(* CoDeSys 2.3.9.41 project: Berdyansl_KNS_bez_zadv.pro *)
(* Libraries: ComService.lib 21.5.09 13:28:28, SysLibCom.lib 20.2.06 12:31:08, ModBus.lib 27.5.09 08:22:38, STANDARD.LIB 4.10.05 10:14:46, IECSFC.LIB 13.4.06 14:51:28, SYSLIBTIME.LIB 20.2.06 12:31:16, SYSTASKINFO.LIB 20.2.06 12:31:38, ANALYZATION.LIB 5.10.99 08:05:06 *)

(* PLC configuration (modules and I/O channels)
DInputs [ID10051] node 0, in %IB0.0 out %QB0.0 {BName = #NДискретные Вх.#A0}
  AT %IB0.0.0 [DInput] Битовая маска входов {CPString128 = #NСост.Дискр.Вх.#Fr.Cn#H2D26#A3#T02#O#B0120#V2; DinLM = #NЛогика Дискр.Вх#Finv.D#B0121#A0#V2#T02#D00#MFF; DinFl = #NПост.Ф.ДребКонт#FTin.F#B0122#A0#U0017#T02#D0A#MFF}
Outputs [ID10057] node 1, in %IB0.1 out %QB0.1 {BName = #NВУ#A0}
  AT %QD0.1.0 [AnalogOutput0] Выход 1 {CPString128 = #NСост.ВУ1#Fr.oe#I00#B0000#A0#O#C3#T00#M+1.00E+00; AoutPWMP = #NПериод ШИМ ВУ1#Fthpd#I00#B0123#A0#U0017#T01#D03E8#L0002#MFDE8; AoutPWMM = #NМин.имп.ШИМ ВУ1#Ft.L#I00#B012B#A0#U0017#T01#D0032#L0001#M1388; AoutSafeValue = #NБезоп.сост.ВУ1#FO.ALr#I00#B0010#A0#C3#T00#D+0.00E+00#M+1.00E+00}
  DO2 AT %QD0.1.1 [AnalogOutput1] Пуск Плавного пуска 2 {CPString128 = #NСост.ВУ2#Fr.oe#HE894#I01#A0#T00#C3#M+1.00E+00#O#B0002; AoutPWMP = #NПериод ШИМ ВУ2#Fthpd#I01#B0124#A0#U0017#T01#D03E8#L0002#MFDE8; AoutPWMM = #NМин.имп.ШИМ ВУ2#Ft.L#I01#B012C#A0#U0017#T01#D0032#L0001#M1388; AoutSafeValue = #NБезоп.сост.ВУ2#FO.ALr#I01#B0012#A0#C3#T00#D+0.00E+00#M+1.00E+00}
  DO3 AT %QD0.1.2 [AnalogOutput2] Пуск Плавного пуска 1 {CPString128 = #NСост.ВУ3#Fr.oe#HE894#I02#A0#T00#C3#M+1.00E+00#O#B0004; AoutPWMP = #NПериод ШИМ ВУ3#Fthpd#I02#B0125#A0#U0017#T01#D03E8#L0002#MFDE8; AoutPWMM = #NМин.имп.ШИМ ВУ3#Ft.L#I02#B012D#A0#U0017#T01#D0032#L0001#M1388; AoutSafeValue = #NБезоп.сост.ВУ3#FO.ALr#I02#B0014#A0#C3#T00#D+0.00E+00#M+1.00E+00}
  DO4 AT %QD0.1.3 [AnalogOutput3] Авария {CPString128 = #NСост.ВУ4#Fr.oe#HE894#I03#A0#T00#C3#M+1.00E+00#O#B0006; AoutPWMP = #NПериод ШИМ ВУ4#Fthpd#I03#B0126#A0#U0017#T01#D03E8#L0002#MFDE8; AoutPWMM = #NМин.имп.ШИМ ВУ4#Ft.L#I03#B012E#A0#U0017#T01#D0032#L0001#M1388; AoutSafeValue = #NБезоп.сост.ВУ4#FO.ALr#I03#B0016#A0#C3#T00#D+0.00E+00#M+1.00E+00}
  DO5 AT %QD0.1.4 [AnalogOutput4] Питание Видеокамеры {CPString128 = #NСост.ВУ5#Fr.oe#HE894#I04#A0#T00#C3#M+1.00E+00#O#B0008; AoutPWMP = #NПериод ШИМ ВУ5#Fthpd#I04#B0127#A0#U0017#T01#D03E8#L0002#MFDE8; AoutPWMM = #NМин.имп.ШИМ ВУ5#Ft.L#I04#B012F#A0#U0017#T01#D0032#L0001#M1388; AoutSafeValue = #NБезоп.сост.ВУ5#FO.ALr#I04#B0018#A0#C3#T00#D+0.00E+00#M+1.00E+00}
  DO6 AT %QD0.1.5 [AnalogOutput5] Управление Дренажным насосом {CPString128 = #NСост.ВУ6#Fr.oe#HE894#I05#A0#T00#C3#M+1.00E+00#O#B000A; AoutPWMP = #NПериод ШИМ ВУ6#Fthpd#I05#B0128#A0#U0017#T01#D03E8#L0002#MFDE8; AoutPWMM = #NМин.имп.ШИМ ВУ6#Ft.L#I05#A0#B0130#U0017#T01#D0032#L0001#M1388; AoutSafeValue = #NБезоп.сост.ВУ6#FO.ALr#I05#B001A#A0#C3#T00#D+0.00E+00#M+1.00E+00}
  DO7 AT %QD0.1.6 [AnalogOutput6] Управление ПЛАВНЫМ ПУСКОМ НАСОСА 2 {CPString128 = #NСост.ВУ7#Fr.oe#HE894#I06#A0#T00#C3#M+1.00E+00#O#B000C; AoutPWMP = #NПериод ШИМ ВУ7#Fthpd#I06#B0129#A0#U0017#T01#D03E8#L0002#MFDE8; AoutPWMM = #NМин.имп.ШИМ ВУ7#Ft.L#I06#B0131#A0#U0017#T01#D0032#L0001#M1388; AoutSafeValue = #NБезоп.сост.ВУ7#FO.ALr#I06#B001C#A0#C3#T00#D+0.00E+00#M+1.00E+00}
  DO8 AT %QD0.1.7 [AnalogOutput7] Управление ПЛАВНЫМ ПУСКОМ НАСОСА 1 {CPString128 = #NСост.ВУ8#Fr.oe#HE894#I07#A0#T00#C3#M+1.00E+00#O#B000E; AoutPWMP = #NПериод ШИМ ВУ8#Fthpd#I07#B012A#A0#U0017#T01#D03E8#L0002#MFDE8; AoutPWMM = #NМин.имп.ШИМ ВУ8#Ft.L#I07#A0#B0132#U0017#T01#D0032#L0001#M1388; AoutSafeValue = #NБезоп.сост.ВУ8#FO.ALr#I07#B001E#A0#C3#T00#D+0.00E+00#M+1.00E+00}
AInputs [ID10055] node 2, in %IB0.2 out %QB0.2 {BName = #NАналоговые Вх.#A0; Spay = #NКоррекция ХС#Fcj-.c#B0133#A0#U002A#T03#D01}
  AT %ID0.2.0 [AnalogInput0] Аналоговый вход 1 {CPString128 = #NДатчик уровня#Fread#H8784#I00#A3#T10#C2#O#B0020#V3; AinType = #NТип датчика 1#Fin-t#H932D#I00#A0#U002F#T04#D10#M15#B0134; InFD = #NПост. фильтра 1#Fin.Fd#I00#B013C#A0#U0018#T01#D0005#M0708; InFG = #NПолоса Фильтра1#Fin.FG#I00#B0030#A0#T00#D+1.00E+01#L+0.00E+01#M+9.99E+03}
  AT %ID0.2.1 [AnalogInputTime0] Время измерения 1
  AI AT %ID0.2.2 [AnalogInput1] Аналоговый вход 2 {CPString128 = #NДатчик давления#Fread#H8784#I01#A3#T10#C2#O#B0022#V3; AinType = #NДатчик уровня#Fin-t#H932D#I01#A0#U002F#T04#D10#M15#B0135; InFD = #NПост. фильтра 2#Fin.Fd#H1659#I01#A0#U0018#T01#D0005#M0708#B013D; InFG = #NПолоса Фильтра2#Fin.FG#I01#B0032#A0#T00#D+1.00E+01#L+0.00E+01#M+9.99E+03}
  AT %ID0.2.3 [AnalogInputTime1] Время измерения 2
  AT %ID0.2.4 [AnalogInput2] Аналоговый вход 3 {CPString128 = #NВход 3#Fread#H8784#I02#A3#T10#C2#O#B0024#V3; AinType = #NТип датчика 3#Fin-t#H932D#I02#A0#U002F#T04#D00#M15#B0136; InFD = #NПост. фильтра 3#Fin.Fd#I02#B013E#A0#U0018#T01#D0005#M0708; InFG = #NПолоса Фильтра3#Fin.FG#I02#B0034#A0#T00#D+1.00E+01#L+0.00E+01#M+9.99E+03}
  AT %ID0.2.5 [AnalogInputTime2] Время измерения 3
  AT %ID0.2.6 [AnalogInput3] Аналоговый вход 4 {CPString128 = #NВход 4#Fread#H8784#I03#A3#T10#C2#O#B0026#V3; AinType = #NТип датчика 4#Fin-t#H932D#I03#A0#U002F#T04#D00#M15#B0137; InFD = #NПост. фильтра 4#Fin.Fd#I03#B013F#A0#U0018#T01#D0005#M0708; InFG = #NПолоса Фильтра4#Fin.FG#I03#A0#B0036#T00#D+1.00E+01#L+0.00E+01#M+9.99E+03}
  AT %ID0.2.7 [AnalogInputTime3] Время измерения 4
  AT %ID0.2.8 [AnalogInput4] Аналоговый вход 5 {CPString128 = #NВход 5#Fread#H8784#I04#A3#T10#C2#O#B0028#V3; AinType = #NТип датчика 5#Fin-t#H932D#I04#A0#U002F#T04#D00#M15#B0138; InFD = #NПост. фильтра 5#Fin.Fd#I04#B0140#A0#U0018#T01#D0005#M0708; InFG = #NПолоса Фильтра5#Fin.FG#I04#B0038#A0#T00#D+1.00E+01#L+0.00E+01#M+9.99E+03}
  AT %ID0.2.9 [AnalogInputTime4] Время измерения 5
  AT %ID0.2.10 [AnalogInput5] Аналоговый вход 6 {CPString128 = #NВход 6#Fread#H8784#I05#A3#T10#C2#O#B002A#V3; AinType = #NТип датчика 6#Fin-t#H932D#I05#A0#U002F#T04#D00#M15#B0139; InFD = #NПост. фильтра 6#Fin.Fd#I05#B0141#A0#U0018#T01#D0005#M0708; InFG = #NПолоса Фильтра6#Fin.FG#I05#B003A#A0#T00#D+1.00E+01#L+0.00E+01#M+9.99E+03}
  AT %ID0.2.11 [AnalogInputTime5] Время измерения 6
  AT %ID0.2.12 [AnalogInput6] Аналоговый вход 7 {CPString128 = #NВход 7#Fread#H8784#I06#A3#T10#C2#O#B002C#V3; AinType = #NТип датчика 7#Fin-t#H932D#I06#A0#U002F#T04#D00#M15#B013A; InFD = #NПост. фильтра 7#Fin.Fd#I06#B0142#A0#U0018#T01#D0005#M0708; InFG = #NПолоса Фильтра7#Fin.FG#I06#B003C#A0#T00#D+1.00E+01#L+0.00E+01#M+9.99E+03}
  AT %ID0.2.13 [AnalogInputTime6] Время измерения 7
  AT %ID0.2.14 [AnalogInput7] Аналоговый вход 8 {CPString128 = #NВход 8#Fread#H8784#I07#A3#T10#C2#O#B002E#V3; AinType = #NТип датчика 8#Fin-t#H932D#I07#A0#U002F#T04#D00#M15#B013B; InFD = #NПост. фильтра 8#Fin.Fd#I07#B0143#A0#U0018#T01#D0005#M0708; InFG = #NПолоса Фильтра8#Fin.FG#I07#B003E#A0#T00#D+1.00E+01#L+0.00E+01#M+9.99E+03}
  AT %ID0.2.15 [AnalogInputTime7] Время измерения 8
MR1_Outputs [ID10053] node 3, in %IB0.3 out %QB0.3 {BName = #NВУ МР1#A0}
  AT %QB0.3.0 [DOutput] ВУ МР1 {CPString128 = #NСост.ВУ МР1#Fr.oe.s#B0144#A0#O#V2#T02}
Additional [ID10059] node 4, in %IB0.4 out %QB0.4 {BName = #NДоп.пар-ры#A0}
  Illumination AT %QB0.4.0 [LCDLight] Подсветка {CPString128 = #NЯрк.подсв.ЖКИ#Find.i#H1845#A0#T02#D2D#M32#B0145}
  AT %QB0.4.1 [LCDContrast] Контраст {CPString128 = #NКонтраст ЖКИ#Find.C#H074A#A0#T02#D19#M20#L05#B0146}
  Keyboard AT %IW0.4.2 [KBD] Клавиатура {CPString128 = #NСост.клавиатуры#Fkbrd#H399B#A3#T02#O#B0147; KBDBeep = #NЗвук кнопок#Fbeep#B0148#A0#U002A#T03#D01}
  Clock AT %QD0.4.3 [RTS] Часы контроллера {RTSPar = #NВремя и дата#FrtC#HFA30#A0#T05#O#B0040}
  Svetodiod AT %QB0.4.4 [LED] Светодиоды {CPString128 = #NСос.светодиодов#Find.L#HF304#A0#T02#D00#M3F#L00#O#B0149#V2}
Versions [ID10060] node 5, in %IB0.5 out %QB0.5 {BName = #NВерсииПрошивок#A0}
  AT %QB0.5.0 [DevName] Имя устройства {CPString128 = #NИмя устройства#Fdev#B0042#A3#O#T08}
  AT %IB0.5.1 [HardVer] Прошивка {CPString128 = #NВерсия прошивки#Fver#B004A#A3#O#T08}
  AT %QB0.5.2 [SoftVer] Программа {CPString128 = #NВерсияПрограммы#Fp.ver#B0052#A3#O#T08}
RS-1 [ID10061] node 6, in %IB0.6 out %QB0.6 {BName = #NНастр.RS-1#A0; RSBPS = #NСкорость#FbPS#I00#B014A#A0#U0046#T04#D00#M09; RSWLen = #NДлина слова#FLen#I00#B014B#A0#U0005#T04#D03#M03; RSPrt = #NЧётность#Fprty#I00#B014C#A0#U009A#T04#D04#M04; RSStp = #NСтоп биты#Fsbit#I00#B014D#A0#U00A1#T04#D00#M02; RSALen = #NДлина адреса#Fa.len#I00#B014E#A0#U0055#T03#D00; RSAdr = #NАдрес прибора#FAddr#I00#B014F#A0#T01#D0010#M07FF; RSDl = #NЗадержка ответа#FRs.dl#I00#B0150#A0#U0017#T02#D05#M32}
RS-2 [ID10062] node 7, in %IB0.7 out %QB0.7 {BName = #NНастр.RS-2#A0; RSBPS = #NСкорость#FbPS#I01#B0151#A0#U0046#T04#D00#M09; RSWLen = #NДлина слова#FLen#I01#B0152#A0#U0005#T04#D03#M03; RSPrt = #NЧётность#Fprty#I01#B0153#A0#U009A#T04#D04#M04; RSStp = #NСтоп биты#Fsbit#I01#B0154#A0#U00A1#T04#D00#M02; RSALen = #NДлина адреса#Fa.len#I01#B0155#A0#U0055#T03#D00; RSAdr = #NАдрес прибора#FAddr#I01#B0156#A0#T01#D0010#M07FF; RSDl = #NЗадержка ответа#FRs.dl#I01#B0157#A0#U0017#T02#D05#M32}
WorkInd [ID10100] node 1, in %IB1 out %QB1 {WIChanelCount = 6}
SubMenu [ID11000] node 2, in %IB2 out %QB2 {BName = #NВетка#A0}
  SubMenu [ID11000] node 0, in %IB2.0 out %QB2.0 {BName = #NВетка#A0}
ATS22_1_p84 AT %QX2.0.0.0 [BoolPar] Канал управления Mb\клемник {CPString128 = #NБулевский#A0#U00AA#T03#D00}
ATS22_1_p752b3 AT %QX2.0.1.0 [BoolPar] Сброс Аварии {CPString128 = #NБулевский#A0#U00AA#T03#D00}
SubMenu [ID11000] node 1, in %IB2.1 out %QB2.1 {BName = #NВетка#A0}
mb_in1 AT %QX2.1.0.0 [BoolPar] {CPString128 = #NБулевский#A0#U00AA#T03#D00#O}
mb_in2 AT %QX2.1.1.0 [BoolPar] {CPString128 = #NБулевский#A0#U00AA#T03#D00#O}
mb_in3 AT %QX2.1.2.0 [BoolPar] {CPString128 = #NБулевский#A0#U00AA#T03#D00#O}
mb_in4 AT %QX2.1.3.0 [BoolPar] {CPString128 = #NБулевский#A0#U00AA#T03#D00#O}
mb_in5 AT %QX2.1.4.0 [BoolPar] {CPString128 = #NБулевский#A0#U00AA#T03#D00}
mb_in6 AT %QX2.1.5.0 [BoolPar] {CPString128 = #NБулевский#A0#U00AA#T03#D00}
mb_in7 AT %QX2.1.6.0 [BoolPar] {CPString128 = #NБулевский#A0#U00AA#T03#D00}
mb_in8 AT %QX2.1.7.0 [BoolPar] {CPString128 = #NБулевский#A0#U00AA#T03#D00}
mb_in9 AT %QX2.1.8.0 [BoolPar] {CPString128 = #NБулевский#A0#U00AA#T03#D00}
mb_in10 AT %QX2.1.9.0 [BoolPar] {CPString128 = #NБулевский#A0#U00AA#T03#D00}
mb_in11 AT %QX2.1.10.0 [BoolPar] {CPString128 = #NБулевский#A0#U00AA#T03#D00}
mb_in12 AT %QX2.1.11.0 [BoolPar] {CPString128 = #NБулевский#A0#U00AA#T03#D00}
mb_in13 AT %QX2.1.12.0 [BoolPar] Контроль доступа Датч 1 {CPString128 = #NБулевский#A0#U00AA#T03#D00}
mb_in14 AT %QX2.1.13.0 [BoolPar] {CPString128 = #NБулевский#A0#U00AA#T03#D00}
mb_in15 AT %QX2.1.14.0 [BoolPar] {CPString128 = #NБулевский#A0#U00AA#T03#D00}
mb_in16 AT %QX2.1.15.0 [BoolPar] {CPString128 = #NБулевский#A0#U00AA#T03#D00}
mb_in17 AT %QX2.1.16.0 [BoolPar] {CPString128 = #NБулевский#A0#U00AA#T03#D00}
mb_in18 AT %QX2.1.17.0 [BoolPar] {CPString128 = #NБулевский#A0#U00AA#T03#D00}
mb_in19 AT %QX2.1.18.0 [BoolPar] {CPString128 = #NБулевский#A0#U00AA#T03#D00}
mb_in20 AT %QX2.1.19.0 [BoolPar] {CPString128 = #NБулевский#A0#U00AA#T03#D00}
mb_in21 AT %QX2.1.20.0 [BoolPar] {CPString128 = #NБулевский#A0#U00AA#T03#D00}
mb_in22 AT %QX2.1.21.0 [BoolPar] {CPString128 = #NБулевский#A0#U00AA#T03#D00}
mb_in23 AT %QX2.1.22.0 [BoolPar] {CPString128 = #NБулевский#A0#U00AA#T03#D00}
mb_in24 AT %QX2.1.23.0 [BoolPar] {CPString128 = #NБулевский#A0#U00AA#T03#D00}
%Mmb_in25 AT %QX2.1.24.0 [BoolPar] {CPString128 = #NБулевский#A0#U00AA#T03#D00}
mb_in26 AT %QX2.1.25.0 [BoolPar] {CPString128 = #NБулевский#A0#U00AA#T03#D00}
mb_in27 AT %QX2.1.26.0 [BoolPar] {CPString128 = #NБулевский#A0#U00AA#T03#D00}
mb_in28 AT %QX2.1.27.0 [BoolPar] {CPString128 = #NБулевский#A0#U00AA#T03#D00}
mb_in29 AT %QX2.1.28.0 [BoolPar] {CPString128 = #NБулевский#A0#U00AA#T03#D00}
mb_in30 AT %QX2.1.29.0 [BoolPar] {CPString128 = #NБулевский#A0#U00AA#T03#D00}
mb_in31 AT %QX2.1.30.0 [BoolPar] {CPString128 = #NБулевский#A0#U00AA#T03#D00}
mb_in32 AT %QX2.1.31.0 [BoolPar] {CPString128 = #NБулевский#A0#U00AA#T03#D00}
ATS22_2_p84 AT %QX2.2.0.0 [BoolPar] Канал управления Mb\клемник {CPString128 = #NБулевский#A0#U00AA#T03#D00}
ATS22_2_p752b3 AT %QX2.2.1.0 [BoolPar] Сброс Аварии {CPString128 = #NБулевский#A0#U00AA#T03#D00}
ubz_1_p100 AT %QW3.0.0.0 [IntPar] Ток А {CPString128 = #NЦелое#A0#T01#D0000}
ubz_1_p101 AT %QW3.0.1.0 [IntPar] Ток В {CPString128 = #NЦелое#A0#T01#D0000}
ubz_1_p102 AT %QW3.0.2.0 [IntPar] Ток С {CPString128 = #NЦелое#A0#T01#D0000}
ubz_1_p103 AT %QW3.0.3.0 [IntPar] Ток нулевой последовательности {CPString128 = #NЦелое#A0#T01#D0000}
ubz_1_p113 AT %QW3.0.4.0 [IntPar] {CPString128 = #NЦелое#A0#T01#D0000}
ubz_1_p114 AT %QW3.0.5.0 [IntPar] {CPString128 = #NЦелое#A0#T01#D0000}
ubz_1_p115 AT %QW3.0.6.0 [IntPar] {CPString128 = #NЦелое#A0#T01#D0000}
ubz_1_p116 AT %QW3.0.7.0 [IntPar] {CPString128 = #NЦелое#A0#T01#D0000}
ubz_1_p117 AT %QW3.0.8.0 [IntPar] Линейное напряжение А {CPString128 = #NЦелое#A0#T01#D0000}
ubz_1_p118 AT %QW3.0.9.0 [IntPar] {CPString128 = #NЦелое#A0#T01#D0000}
ubz_1_p119 AT %QW3.0.10.0 [IntPar] {CPString128 = #NЦелое#A0#T01#D0000}
ubz_1_p120 AT %QW3.0.11.0 [IntPar] {CPString128 = #NЦелое#A0#T01#D0000}
ubz_1_p121 AT %QW3.0.12.0 [IntPar] {CPString128 = #NЦелое#A0#T01#D0000}
ubz_1_p122 AT %QW3.0.13.0 [IntPar] {CPString128 = #NЦелое#A0#T01#D0000}
IntP [ID11200] node 14, in %IB3.0.14 out %QB3.0.14
  ubz_1_p241 AT %QW3.0.14.0 [IntPar] {CPString128 = #NЦелое#A0#T01#D0000}
IntP [ID11200] node 15, in %IB3.0.15 out %QB3.0.15
  ubz_1_p242 AT %QW3.0.15.0 [IntPar] {CPString128 = #NЦелое#A0#T01#D0000}
ubz_1_p240 AT %QB3.0.16.0 [BytePar] Регистр состояния УБЗ {CPString128 = #NБайт#A0#T02#D00}
ubz_1_p241_1 AT %QB3.0.17.0 [BytePar] Регистр Аварии 1 {CPString128 = #NБайт#A0#T02#D00}
ubz_1_p241_2 AT %QB3.0.18.0 [BytePar] Регистр Аварии 1 {CPString128 = #NБайт#A0#T02#D00}
ubz_1_p242_1 AT %QB3.0.19.0 [BytePar] Регистр Аварии 2 {CPString128 = #NБайт#A0#T02#D00}
ubz_1_p242_2 AT %QB3.0.20.0 [BytePar] Регистр Аварии 2 {CPString128 = #NБайт#A0#T02#D00}
SubMenu [ID11000] node 1, in %IB3.1 out %QB3.1 {BName = #NВетка#A0}
ubz_2_p100 AT %QW3.1.0.0 [IntPar] Ток А {CPString128 = #NЦелое#A0#T01#D0000}
ubz_2_p101 AT %QW3.1.1.0 [IntPar] Ток В {CPString128 = #NЦелое#A0#T01#D0000}
ubz_2_p102 AT %QW3.1.2.0 [IntPar] Ток С {CPString128 = #NЦелое#A0#T01#D0000}
ubz_2_p103 AT %QW3.1.3.0 [IntPar] Ток нулевой последовательности {CPString128 = #NЦелое#A0#T01#D0000}
ubz_2_p113 AT %QW3.1.4.0 [IntPar] {CPString128 = #NЦелое#A0#T01#D0000}
ubz_2_p114 AT %QW3.1.5.0 [IntPar] {CPString128 = #NЦелое#A0#T01#D0000}
ubz_2_p115 AT %QW3.1.6.0 [IntPar] {CPString128 = #NЦелое#A0#T01#D0000}
ubz_2_p116 AT %QW3.1.7.0 [IntPar] {CPString128 = #NЦелое#A0#T01#D0000}
ubz_2_p117 AT %QW3.1.8.0 [IntPar] Линейное напряжение А {CPString128 = #NЦелое#A0#T01#D0000}
ubz_2_p118 AT %QW3.1.9.0 [IntPar] {CPString128 = #NЦелое#A0#T01#D0000}
ubz_2_p119 AT %QW3.1.10.0 [IntPar] {CPString128 = #NЦелое#A0#T01#D0000}
ubz_2_p120 AT %QW3.1.11.0 [IntPar] {CPString128 = #NЦелое#A0#T01#D0000}
ubz_2_p121 AT %QW3.1.12.0 [IntPar] {CPString128 = #NЦелое#A0#T01#D0000}
ubz_2_p122 AT %QW3.1.13.0 [IntPar] {CPString128 = #NЦелое#A0#T01#D0000}
IntP [ID11200] node 14, in %IB3.1.14 out %QB3.1.14
  ubz_2_p241 AT %QW3.1.14.0 [IntPar] {CPString128 = #NЦелое#A0#T01#D0000}
  ubz_2_p242 AT %QW3.1.15.0 [IntPar] {CPString128 = #NЦелое#A0#T01#D0000}
SubMenu [ID11000] node 2, in %IB3.2 out %QB3.2 {BName = #NВетка#A0}
ATS22_1_p279 AT %QW3.2.0.0 [IntPar] Проследняя неисправность {CPString128 = #NЦелое#A0#T01#D0000}
ATS22_1_p256 AT %QW3.2.1.0 [IntPar] Состояние Плавноо пуска {CPString128 = #NЦелое#A0#T01#D0000}
ATS22_1_p257 AT %QW3.2.2.0 [IntPar] Ток фазы А {CPString128 = #NЦелое#A0#T01#D0000}
ATS22_1_p259 AT %QW3.2.3.0 [IntPar] Ток фазы С {CPString128 = #NЦелое#A0#T01#D0000}
ATS22_1_p258 AT %QW3.2.4.0 [IntPar] Ток фазы В {CPString128 = #NЦелое#A0#T01#D0000}
ATS22_1_p260 AT %QW3.2.5.0 [IntPar] Линейное напряжение {CPString128 = #NЦелое#A0#T01#D0000}
SubMenu [ID11000] node 3, in %IB3.3 out %QB3.3 {BName = #NВетка#A0}
ATS22_2_p279 AT %QW3.3.0.0 [IntPar] {CPString128 = #NЦелое#A0#T01#D0000}
ATS22_2_p256 AT %QW3.3.1.0 [IntPar] {CPString128 = #NЦелое#A0#T01#D0000}
ATS22_2_p257 AT %QW3.3.2.0 [IntPar] {CPString128 = #NЦелое#A0#T01#D0000}
ATS22_2_p259 AT %QW3.3.3.0 [IntPar] {CPString128 = #NЦелое#A0#T01#D0000}
ATS22_2_p258 AT %QW3.3.4.0 [IntPar] {CPString128 = #NЦелое#A0#T01#D0000}
ATS22_2_p260 AT %QW3.3.5.0 [IntPar] {CPString128 = #NЦелое#A0#T01#D0000}
SubMenu [ID11000] node 4, in %IB4 out %QB4 {BName = #NВетка#A0}
*)

(* Global variable list: Global_Variables *)
VAR_GLOBAL
(*+++++++++++++++++++++++++++++++++++++++++++++++++++++++++++++++++++*)
(* переменные Modbus *)
	funcComService:COM_SERVICE;(*экземпляр COM_SERVICE*)
	cmSettings:COMSETTINGS;(* настройки COM- порта *)
	cmpl: BOOL;(* статус выполнения*)
	Buffer:ARRAY[0..255] OF BYTE;								(*буфер данных Modbus*)

(*+++++++++++++++++++++++++++++++++++++++++++++++++++++++++++++++++++*)

(*+++++++++++++++++++++++++++++++++++++++++++++++++++++++++++++++++++*)
(* Переменные плавного пуска №1*)
	Status_UZ1:WORD; (* Состояние плавного пуска №1 *)

(* Переменные плавного пуска №2*)
	Status_UZ2:WORD; (* Состояние плавного пуска №2 *)

(* Переменные УБЗ-302 №1 *)
	Alarm_UBZ1_p241:WORD; (*Аварии двигателя  УБЗ*)
	Alarm_UBZ1_p242:WORD; (*Аварии самого УБЗ*)

END_VAR

(* POU PLC_PRG, ST *)
PROGRAM PLC_PRG
VAR
END_VAR
prgModbus();
END_PROGRAM

(* POU prgModbus, ST *)
PROGRAM prgModbus
VAR

	byMbRequest:BYTE:=0;(* Номер опроса по Мб *)
	funcMbReadHoldRegs:MB_RD_HOLD_REGS;(*Modbus, экземпляр функ. 03, чтение регистров хранения*)
	funcMbReadInpRegs:MB_RD_INP_REGS;(*Modbus, экземпляр функ. 04, чтение регистров ввода*)
	funcMbWriteSngReg:MB_WR_SNG_REG;(*Modbus, экземпляр функ. 06, запись регистра хранения*)
	funcMbWriteRegs:MB_WR_REGS;(*Modbus, экземпляр функ. 16, запись регистров хранения*)


END_VAR
(* Обработка данных Modbus *)
	IF NOT funcComService.ready THEN
		cmSettings.Port:=1;(*номер COM-порта*)
		cmSettings.dwBaudRate:=19200;
		cmSettings.byParity:=0;
		cmSettings.dwTimeout:=0;
		cmSettings.byStopBits:=0;
		cmSettings.dwBufferSize:=0;
		cmSettings.dwScan:=0;
		funcComService(Enable:=TRUE , Settings:=cmSettings , Task:=OPEN_TSK  );
	END_IF

(*=======================================================================*)
(*===========Опрос===============*)
IF funcComService.ready THEN
	CASE byMbRequest OF
(* Опрос UZ1 *)
(*
Add: 1;
ctrl: LCL;
tt: 5.0;
For: 8n1;
tbr 19.2;
*)
    
0:(*считывает значение состояния плавного пуска*)
			funcMbReadHoldRegs(
				Enable:=TRUE ,					(*запустить блок*)
				Mode:=MB_RTU ,				(*режим передачи*)
				DevAddr:=1 ,						(*адрес опрашиваемого устройства*)
				FirstAddr:=256 ,				(*номер регистра*)
				Quantity:=1,						(*количество регистров*)
				ComHandle:=cmSettings.Port ,
				TimeOut:=T#50ms ,				(*таймаут*)
				Buffer:=Buffer);
				IF funcMbReadHoldRegs.Complete THEN
					IF funcMbReadHoldRegs.Exception=0 THEN
						Status_UZ1:=WORD_TO_INT(BYTE_TO_WORD(Buffer[1]) OR SHL(BYTE_TO_WORD(Buffer[0]),8));
						IF Status_UZ1.0=1 THEN ATS22_1_p256:=0; (* 0 - остановлен*)
						ELSIF Status_UZ1.1=1 THEN ATS22_1_p256:=1; (* 1 - запущен*)
						ELSIF Status_UZ1.2=1 THEN ATS22_1_p256:=2; (* 3 -авария*)
						ELSIF Status_UZ1.15=1 THEN ATS22_1_p256:=3; (* 2 - плавный запуск или останов *)
						END_IF
					byMbRequest:=1;
					END_IF
				END_IF
1: (*считывает проследнюю неисправность *)
			funcMbReadHoldRegs(
				Enable:=TRUE ,					(*запустить блок*)
				Mode:=MB_RTU ,					(*режим передачи*)
				DevAddr:=1 ,						(*адрес опрашиваемого устройства*)
				FirstAddr:=279,					(*номер регистра*)
				Quantity:=1,						(*количество регистров*)
				ComHandle:=cmSettings.Port ,
				TimeOut:=T#50ms ,				(*таймаут*)
				Buffer:=Buffer);
				IF funcMbReadHoldRegs.Complete THEN
					IF funcMbReadHoldRegs.Exception=0 THEN
						ATS22_1_p279:=WORD_TO_INT(BYTE_TO_WORD(BUFFER[1]) OR SHL(BYTE_TO_WORD(BUFFER[0]),8));

						byMbRequest:=2;
					END_IF
				END_IF

2: (*считывает Ток фазы А *)
				funcMbReadHoldRegs(
				Enable:=TRUE ,					(*запустить блок*)
				Mode:=MB_RTU ,					(*режим передачи*)
				DevAddr:=1 ,						(*адрес опрашиваемого устройства*)
				FirstAddr:=257,					(*номер регистра*)
				Quantity:=1,						(*количество регистров*)
				ComHandle:=cmSettings.Port ,
				TimeOut:=T#50ms ,				(*таймаут*)
				Buffer:=Buffer);
				IF funcMbReadHoldRegs.Complete THEN
					IF funcMbReadHoldRegs.Exception=0 THEN
					ATS22_1_p257:=WORD_TO_INT(BYTE_TO_WORD(Buffer[1]) OR SHL(BYTE_TO_WORD(Buffer[0]),8));

					byMbRequest:=3;
					END_IF
				END_IF

3: (*считывает Ток фазы B *)
				funcMbReadHoldRegs(
				Enable:=TRUE ,					(*запустить блок*)
				Mode:=MB_RTU ,					(*режим передачи*)
				DevAddr:=1 ,						(*адрес опрашиваемого устройства*)
				FirstAddr:=258,					(*номер регистра*)
				Quantity:=1,						(*количество регистров*)
				ComHandle:=cmSettings.Port ,
				TimeOut:=T#50ms ,				(*таймаут*)
				Buffer:=Buffer);
				IF funcMbReadHoldRegs.Complete THEN
					IF funcMbReadHoldRegs.Exception=0 THEN
					ATS22_1_p258:=WORD_TO_INT(BYTE_TO_WORD(Buffer[1]) OR SHL(BYTE_TO_WORD(Buffer[0]),8));

					byMbRequest:=4;
					END_IF
				END_IF

4:(*считывает Ток фазы C *)
				funcMbReadHoldRegs(
				Enable:=TRUE ,					(*запустить блок*)
				Mode:=MB_RTU ,					(*режим передачи*)
				DevAddr:=1 ,						(*адрес опрашиваемого устройства*)
				FirstAddr:=259,					(*номер регистра*)
				Quantity:=1,						(*количество регистров*)
				ComHandle:=cmSettings.Port ,
				TimeOut:=T#50ms ,				(*таймаут*)
				Buffer:=Buffer);
				IF funcMbReadHoldRegs.Complete THEN
					IF funcMbReadHoldRegs.Exception=0 THEN
					ATS22_1_p259:=WORD_TO_INT(BYTE_TO_WORD(Buffer[1]) OR SHL(BYTE_TO_WORD(Buffer[0]),8));

					byMbRequest:=5;
					END_IF
				END_IF

5:	(*считывает Линейное напряжение *)
				funcMbReadHoldRegs(
				Enable:=TRUE ,					(*запустить блок*)
				Mode:=MB_RTU ,					(*режим передачи*)
				DevAddr:=1 ,						(*адрес опрашиваемого устройства*)
				FirstAddr:=260,					(*номер регистра*)
				Quantity:=1,						(*количество регистров*)
				ComHandle:=cmSettings.Port ,
				TimeOut:=T#50ms ,				(*таймаут*)
				Buffer:=Buffer);
				IF funcMbReadHoldRegs.Complete THEN
					IF funcMbReadHoldRegs.Exception=0 THEN
					ATS22_1_p260:=WORD_TO_INT(BYTE_TO_WORD(Buffer[1]) OR SHL(BYTE_TO_WORD(Buffer[0]),8));

					byMbRequest:=6;
					END_IF
				END_IF

6:	IF ATS22_1_p84 THEN (*перевод в управление по МВ*)

		funcMbWriteSngReg(
				Enable:=TRUE ,					(*запустить блок*)
				Mode:=MB_RTU ,					(*режим передачи*)
				DevAddr:=1 ,						(*адрес опрашиваемого устройства*)
				REGAddr:=84,					(*номер регистра*)
				Value:=1,						 (* Если 1 то управление по modbus *)
				ComHandle:=cmSettings.Port ,
				TimeOut:=T#20ms);
				IF funcMbWriteSngReg.Complete THEN
					byMbRequest:=7;
				END_IF
	ELSE
		funcMbWriteSngReg(
				Enable:=TRUE ,					(*запустить блок*)
				Mode:=MB_RTU ,					(*режим передачи*)
				DevAddr:=1 ,						(*адрес опрашиваемого устройства*)
				REGAddr:=84,					(*номер регистра*)
				Value:=0,						 (* Если 1 то управление по modbus *)
				ComHandle:=cmSettings.Port ,
				TimeOut:=T#20ms);
				IF funcMbWriteSngReg.Complete THEN
					byMbRequest:=7;
				END_IF
	END_IF

7: (*Сброс Аварии ATS22 №1*)
	IF ATS22_1_p752b3 THEN
		funcMbWriteSngReg(
				Enable:=TRUE ,					(*запустить блок*)
				Mode:=MB_RTU ,					(*режим передачи*)
				DevAddr:=1 ,						(*адрес опрашиваемого устройства*)
				REGAddr:=752,					(*номер регистра*)
				Value:=8,						 (* Если 1 то управление по modbus *)
				ComHandle:=cmSettings.Port ,
				TimeOut:=T#20ms);
				IF funcMbWriteSngReg.Complete THEN
					byMbRequest:=8;
				END_IF
	END_IF

(*=======================================================================*)
(* Опрос UZ2 *)
(*
Add: 2;
ctrl: LCL;
tt: 5.0;
For: 8n1;
tbr 19.2;
*)

8:(*считывает значение состояния плавного пуска*)
			funcMbReadHoldRegs(
				Enable:=TRUE ,					(*запустить блок*)
				Mode:=MB_RTU ,				(*режим передачи*)
				DevAddr:=2 ,						(*адрес опрашиваемого устройства*)
				FirstAddr:=256 ,				(*номер регистра*)
				Quantity:=1,						(*количество регистров*)
				ComHandle:=cmSettings.Port ,
				TimeOut:=T#50ms ,				(*таймаут*)
				Buffer:=Buffer);
				IF funcMbReadHoldRegs.Complete THEN
					IF funcMbReadHoldRegs.Exception=0 THEN
						Status_UZ2:=WORD_TO_INT(BYTE_TO_WORD(Buffer[1]) OR SHL(BYTE_TO_WORD(Buffer[0]),8));
						IF Status_UZ2.0=1 THEN ATS22_2_p256:=0; (* 0 - остановлен*)
						ELSIF Status_UZ2.1=1 THEN ATS22_2_p256:=1; (* 1 - запущен*)
						ELSIF Status_UZ2.2=1 THEN ATS22_2_p256:=2; (* 3 -авария*)
						ELSIF Status_UZ2.15=1 THEN ATS22_2_p256:=3; (* 2 - плавный запуск или останов *)
						END_IF
					byMbRequest:=9;
					END_IF
				END_IF
9: (*считывает проследнюю неисправность *)
			funcMbReadHoldRegs(
				Enable:=TRUE ,					(*запустить блок*)
				Mode:=MB_RTU ,					(*режим передачи*)
				DevAddr:=2 ,						(*адрес опрашиваемого устройства*)
				FirstAddr:=279,					(*номер регистра*)
				Quantity:=1,						(*количество регистров*)
				ComHandle:=cmSettings.Port ,
				TimeOut:=T#50ms ,				(*таймаут*)
				Buffer:=Buffer);
				IF funcMbReadHoldRegs.Complete THEN
					IF funcMbReadHoldRegs.Exception=0 THEN
						ATS22_2_p279:=WORD_TO_INT(BYTE_TO_WORD(BUFFER[1]) OR SHL(BYTE_TO_WORD(BUFFER[0]),8));

						byMbRequest:=10;
					END_IF
				END_IF

10: (*считывает Ток фазы А *)
				funcMbReadHoldRegs(
				Enable:=TRUE ,					(*запустить блок*)
				Mode:=MB_RTU ,					(*режим передачи*)
				DevAddr:=2 ,						(*адрес опрашиваемого устройства*)
				FirstAddr:=257,					(*номер регистра*)
				Quantity:=1,						(*количество регистров*)
				ComHandle:=cmSettings.Port ,
				TimeOut:=T#50ms ,				(*таймаут*)
				Buffer:=Buffer);
				IF funcMbReadHoldRegs.Complete THEN
					IF funcMbReadHoldRegs.Exception=0 THEN
					ATS22_2_p257:=WORD_TO_INT(BYTE_TO_WORD(Buffer[1]) OR SHL(BYTE_TO_WORD(Buffer[0]),8));

					byMbRequest:=11;
					END_IF
				END_IF

11: (*считывает Ток фазы B *)
				funcMbReadHoldRegs(
				Enable:=TRUE ,					(*запустить блок*)
				Mode:=MB_RTU ,					(*режим передачи*)
				DevAddr:=2 ,						(*адрес опрашиваемого устройства*)
				FirstAddr:=258,					(*номер регистра*)
				Quantity:=1,						(*количество регистров*)
				ComHandle:=cmSettings.Port ,
				TimeOut:=T#50ms ,				(*таймаут*)
				Buffer:=Buffer);
				IF funcMbReadHoldRegs.Complete THEN
					IF funcMbReadHoldRegs.Exception=0 THEN
					ATS22_2_p258:=WORD_TO_INT(BYTE_TO_WORD(Buffer[1]) OR SHL(BYTE_TO_WORD(Buffer[0]),8));

					byMbRequest:=12;
					END_IF
				END_IF

12:(*считывает Ток фазы C *)
				funcMbReadHoldRegs(
				Enable:=TRUE ,					(*запустить блок*)
				Mode:=MB_RTU ,					(*режим передачи*)
				DevAddr:=2 ,						(*адрес опрашиваемого устройства*)
				FirstAddr:=259,					(*номер регистра*)
				Quantity:=1,						(*количество регистров*)
				ComHandle:=cmSettings.Port ,
				TimeOut:=T#50ms ,				(*таймаут*)
				Buffer:=Buffer);
				IF funcMbReadHoldRegs.Complete THEN
					IF funcMbReadHoldRegs.Exception=0 THEN
					ATS22_2_p259:=WORD_TO_INT(BYTE_TO_WORD(Buffer[1]) OR SHL(BYTE_TO_WORD(Buffer[0]),8));

					byMbRequest:=13;
					END_IF
				END_IF

13:	(*считывает Линейное напряжение *)
				funcMbReadHoldRegs(
				Enable:=TRUE ,					(*запустить блок*)
				Mode:=MB_RTU ,					(*режим передачи*)
				DevAddr:=2 ,						(*адрес опрашиваемого устройства*)
				FirstAddr:=260,					(*номер регистра*)
				Quantity:=1,						(*количество регистров*)
				ComHandle:=cmSettings.Port ,
				TimeOut:=T#50ms ,				(*таймаут*)
				Buffer:=Buffer);
				IF funcMbReadHoldRegs.Complete THEN
					IF funcMbReadHoldRegs.Exception=0 THEN
					ATS22_2_p260:=WORD_TO_INT(BYTE_TO_WORD(Buffer[1]) OR SHL(BYTE_TO_WORD(Buffer[0]),8));

					byMbRequest:=14;
					END_IF
				END_IF

14:	IF ATS22_2_p84 THEN (*перевод в управление по МВ*)

		funcMbWriteSngReg(
				Enable:=TRUE ,					(*запустить блок*)
				Mode:=MB_RTU ,					(*режим передачи*)
				DevAddr:=2 ,						(*адрес опрашиваемого устройства*)
				REGAddr:=84,					(*номер регистра*)
				Value:=1,						 (* Если 1 то управление по modbus *)
				ComHandle:=cmSettings.Port ,
				TimeOut:=T#20ms);
				IF funcMbWriteSngReg.Complete THEN
					byMbRequest:=15;
				END_IF
	ELSE
		funcMbWriteSngReg(
				Enable:=TRUE ,					(*запустить блок*)
				Mode:=MB_RTU ,					(*режим передачи*)
				DevAddr:=2 ,						(*адрес опрашиваемого устройства*)
				REGAddr:=84,					(*номер регистра*)
				Value:=0,						 (* Если 1 то управление по modbus *)
				ComHandle:=cmSettings.Port ,
				TimeOut:=T#20ms);
				IF funcMbWriteSngReg.Complete THEN
					byMbRequest:=15;
				END_IF
	END_IF

15: (*Сброс Аварии ATS22 №2*)
	IF ATS22_2_p752b3 THEN
		funcMbWriteSngReg(
				Enable:=TRUE ,					(*запустить блок*)
				Mode:=MB_RTU ,					(*режим передачи*)
				DevAddr:=2 ,						(*адрес опрашиваемого устройства*)
				REGAddr:=752,					(*номер регистра*)
				Value:=8,						 (* Если 1 то управление по modbus *)
				ComHandle:=cmSettings.Port ,
				TimeOut:=T#20ms);
				IF funcMbWriteSngReg.Complete THEN
					byMbRequest:=16;
				END_IF
	END_IF
(*=======================================================================*)
(* Опрос УБЗ-302 №1 *)
(*
Add: 3;
tt: 5.0;
For: 8n1;
tbr 19.2;
*)
16: (* читаем регистры 100....103*)
		funcMbReadHoldRegs(
				Enable:=TRUE ,					(*запустить блок*)
				Mode:=MB_RTU ,					(*режим передачи*)
				DevAddr:=3 ,						(*адрес опрашиваемого устройства*)
				FirstAddr:=100,					(*номер регистра*)
				Quantity:=4,						(*количество регистров*)
				ComHandle:=cmSettings.Port ,
				TimeOut:=T#50ms ,				(*таймаут*)
				Buffer:=Buffer);
				IF funcMbReadHoldRegs.Complete THEN
					IF funcMbReadHoldRegs.Exception=0 THEN
						ubz_1_p100:=WORD_TO_INT(BYTE_TO_WORD(BUFFER[1]) OR SHL(BYTE_TO_WORD(BUFFER[0]),8));(* Ток А *)
						ubz_1_p101:=WORD_TO_INT(BYTE_TO_WORD(BUFFER[3]) OR SHL(BYTE_TO_WORD(BUFFER[2]),8));(* Ток B *)
						ubz_1_p102:=WORD_TO_INT(BYTE_TO_WORD(BUFFER[5]) OR SHL(BYTE_TO_WORD(BUFFER[4]),8));(* Ток С*)
						ubz_1_p103:=WORD_TO_INT(BYTE_TO_WORD(BUFFER[7]) OR SHL(BYTE_TO_WORD(BUFFER[6]),8));(* Ток нулевой последовательности *)
					byMbRequest:=17;
					END_IF
				END_IF

17: (* читаем регистры 113....122*)
		funcMbReadHoldRegs(
				Enable:=TRUE ,					(*запустить блок*)
				Mode:=MB_RTU ,					(*режим передачи*)
				DevAddr:=3 ,						(*адрес опрашиваемого устройства*)
				FirstAddr:=100,					(*номер регистра*)
				Quantity:=4,						(*количество регистров*)
				ComHandle:=cmSettings.Port ,
				TimeOut:=T#50ms ,				(*таймаут*)
				Buffer:=Buffer);
				IF funcMbReadHoldRegs.Complete THEN
					IF funcMbReadHoldRegs.Exception=0 THEN
						ubz_1_p113:=WORD_TO_INT(BYTE_TO_WORD(BUFFER[1]) OR SHL(BYTE_TO_WORD(BUFFER[0]),8));(* Ток обратной последовательности *)
						ubz_1_p114:=WORD_TO_INT(BYTE_TO_WORD(BUFFER[3]) OR SHL(BYTE_TO_WORD(BUFFER[2]),8));(* Фазные напряжение *)
						ubz_1_p115:=WORD_TO_INT(BYTE_TO_WORD(BUFFER[5]) OR SHL(BYTE_TO_WORD(BUFFER[4]),8));
						ubz_1_p116:=WORD_TO_INT(BYTE_TO_WORD(BUFFER[7]) OR SHL(BYTE_TO_WORD(BUFFER[6]),8));
						ubz_1_p117:=WORD_TO_INT(BYTE_TO_WORD(BUFFER[9]) OR SHL(BYTE_TO_WORD(BUFFER[8]),8));(* линейные напряжения *)
						ubz_1_p118:=WORD_TO_INT(BYTE_TO_WORD(BUFFER[11]) OR SHL(BYTE_TO_WORD(BUFFER[10]),8));
						ubz_1_p119:=WORD_TO_INT(BYTE_TO_WORD(BUFFER[13]) OR SHL(BYTE_TO_WORD(BUFFER[12]),8));
						ubz_1_p120:=WORD_TO_INT(BYTE_TO_WORD(BUFFER[15]) OR SHL(BYTE_TO_WORD(BUFFER[14]),8));(* напряжение прямое*)
						ubz_1_p121:=WORD_TO_INT(BYTE_TO_WORD(BUFFER[17]) OR SHL(BYTE_TO_WORD(BUFFER[16]),8));(* напряжение обратное *)
						ubz_1_p122:=WORD_TO_INT(BYTE_TO_WORD(BUFFER[19]) OR SHL(BYTE_TO_WORD(BUFFER[20]),8));(* напряжение нулевой последовательности *)
					byMbRequest:=18;
					END_IF
				END_IF

18: (* Считываем регистры аварий (240 код состояния, 241 авариии двигателя, 242-аварии убз ) *)
			funcMbReadHoldRegs(
				Enable:=TRUE ,					(*запустить блок*)
				Mode:=MB_RTU ,					(*режим передачи*)
				DevAddr:=3 ,						(*адрес опрашиваемого устройства*)
				FirstAddr:=240,					(*номер регистра*)
				Quantity:=2,						(*количество регистров*)
				ComHandle:=cmSettings.Port ,
				TimeOut:=T#50ms ,				(*таймаут*)
				Buffer:=Buffer);
			IF funcMbReadHoldRegs.Complete THEN
				IF funcMbReadHoldRegs.Exception=0 THEN
					ubz_1_p240:=BUFFER[0]; (* состояние убз*)
					ubz_1_p241_1:=buffer[2];(* регистры кодов аварий дввигателя*)
					ubz_1_p241_2:=buffer[3];
					ubz_1_p242_1:=buffer[4];(* регистры кодов аварий УБЗ*)
					ubz_1_p242_2:=buffer[5];
				byMbRequest:=19;
				END_IF
			END_IF



	END_CASE
END_IF
END_PROGRAM
